FUNCTION_BLOCK AxisJogTestSuite EXTENDS TestSuite<TestSuiteParameter.MaxTestCount>
VAR
	StubAxis : AXIS_REF;
	iStubTask : I_Task;
	TestAxisJog : JogBehaviour(stubaxis);
END_VAR

END_FUNCTION_BLOCK

(* stored: Version 1.1.0.1
   POU AxisJogTestSuite: Id {d58fdfa9-a16a-4795-9564-e1d5a0ea8323}, SpecialFunc None *)
